# EPICS autosave request: iocBoot/ioc13LabJackT8_2/auto_settings.req
file "LabJack_T7_settings.req", P=$(P)
file "scan_settings.req",       P=$(P), S=scan1
file "scan_settings.req",       P=$(P), S=scan2
file "scan_settings.req",       P=$(P), S=scan3
file "scan_settings.req",       P=$(P), S=scan4
file "pid_control_settings.req" P=$(P), PID=PID1
file "calc_GSECARS.req",        P=$(P)
